{attribute addProperty BoxType "EL3201-0030-0022"}
{attribute addProperty Id "RTDAT %I*RTD_B51B79FC8110.1250WcStateAT %I*WcState_98A4DF7520.250InfoDataAT %I*InfoData_BC63D37F80100"}
{attribute addProperty CRC "1345030220"}
{attribute addProperty SizeInBites "163"}
{attribute addProperty SizeInBytes "20.375"}
TYPE EL3201_73D65BA5 :
STRUCT
	{attribute addProperty Name "RTD"}
	RTD : RTD_B51B79FC;
	{attribute addProperty Name "WcState"}
	WcState : WcState_98A4DF75;
	{attribute addProperty Name "InfoData"}
	InfoData : InfoData_BC63D37F;
END_STRUCT
END_TYPE

(* stored: Version 1.2.0.0, ProductVersion 3.1.4024.9
   DUT EL3201_73D65BA5: Id {2023a559-6937-477c-8090-47699f50dfee} *)
